FUNCTION_BLOCK PUBLIC Recipe2
VAR_INPUT
	ExecutingRecipe2: BOOL;
	SuccesfullyEnded2: BOOL := FALSE;
END_VAR
VAR_OUTPUT
	SuccesfullyEnded: BOOL := FALSE;
END_VAR
VAR
	State: INT := 0;
	
	MinRotationPosition: INT := 0;
	InitialRotationPosition: INT := 140;
	
	MinLiftingPosition: INT := 0;
	InitialLiftingPosition: INT := 200;
	WoodInitialLiftingPosition: INT := 90;
	
	MinGripPosition: INT := 0;
	MaxGripPosition: INT := 160;

	MotorDirectionEnum: MovementDirection;	// for better clarity on the direction 0 and 1
	MovementEnum: Movement;	// for better clarity on the ON/OFF movement of the motors
END_VAR

IF ExecutingRecipe2 AND (NOT SuccesfullyEnded2) THEN	// we start executing recipe2 (again)
	SuccesfullyEnded := FALSE;
END_IF

IF NOT IO.Switch AND (NOT SuccesfullyEnded2) THEN
	
	IF State = 0 THEN
		State := Rotation(InitialRotationPosition, State);
		
	ELSIF State = 1 THEN
		State := Lifting(InitialLiftingPosition, State);
		
	ELSIF State = 2 THEN
		State := Grip(MaxGripPosition, State);
		
	ELSIF State = 3 THEN
		State := Lifting(MinLiftingPosition, State);
		
	ELSIF State = 4 THEN
		State := Rotation(MinRotationPosition, State);
		
	ELSIF State = 5 THEN
		State := Lifting(WoodInitialLiftingPosition, State);

	ELSIF State = 6 THEN
		State := Grip(MinGripPosition, State);
	
	ELSIF State = 7 THEN
		IO.Initialized := FALSE;
		SuccesfullyEnded := TRUE;
		State := 0;
		RETURN;
	END_IF
END_IF

END_FUNCTION_BLOCK

(* stored: Version 1.1.0.1, ProductVersion 3.1.4024.13
   POU Recipe2: Id {cefbc20c-159f-4896-912e-87a831f8ea44}, SpecialFunc None *)
